PROGRAM SR_Push_and_pick_ITF
VAR
	fbFIFO : FB_FIFO_OOP;
	fbPusher : FB_Pusher_Itf;
	xPush  : BOOL;
	fbPicker  : FB_Picker_Itf;
	xPick  : BOOL;
END_VAR

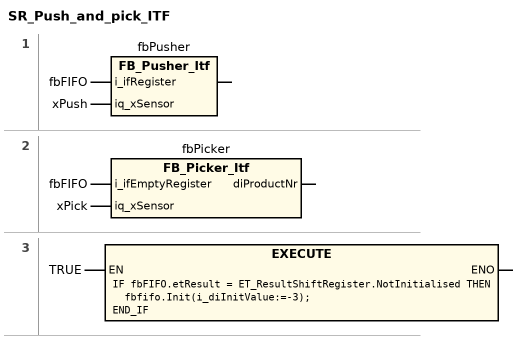
// NETWORK 1
fbPusher(i_ifRegister := fbFIFO, iq_xSensor := xPush); // FB_Pusher_Itf

// NETWORK 2
fbPicker(i_ifEmptyRegister := fbFIFO, iq_xSensor := xPick); // FB_Picker_Itf

// NETWORK 3
IF fbFIFO.etResult = ET_ResultShiftRegister.NotInitialised THEN
	fbfifo.Init(i_diInitValue:=-3);
END_IF

END_PROGRAM

(* stored: Version 1.1.0.1
   POU SR_Push_and_pick_ITF: Id {3bb3a4f7-7d61-476a-b623-3070f8d60c80}, SpecialFunc None *)
